INTERFACE ITF_BaseSaM

METHOD PUBLIC GetMode : E_BaseMachineMode
VAR_INPUT
END_VAR
END_METHOD

METHOD PUBLIC GetState : E_BaseMachineState
VAR_INPUT
END_VAR
END_METHOD

(*			
	EVERDE sp. z o.o.
	Rafał Osajda		25.10.2025		TC 4024.66
	Czy trwa zmianay trybu
*)
METHOD PUBLIC IsChangeModeBusy : BOOL
VAR_INPUT
END_VAR
END_METHOD

(*			
	EVERDE sp. z o.o.
	Rafał Osajda		25.10.2025		TC 4024.66
	Czy trwa zmiana stanu
*)
METHOD PUBLIC IsChangeStateBusy : BOOL
VAR_INPUT

END_VAR
END_METHOD

END_INTERFACE

(* stored: Version 1.1.0.1
   Itf ITF_BaseSaM: Id {e06ea4d8-10a4-07fe-0bda-c5cd43560d4e}
   Method GetMode: Id {17ad96f9-f8c6-06b4-06e2-cdfe42403acb}
   Method GetState: Id {d5368088-86fd-0411-1ca9-12bdae93bf00}
   Method IsChangeModeBusy: Id {0dd216ea-27b5-01b9-033f-72faa5a0d597}
   Method IsChangeStateBusy: Id {2bd79ff5-9782-015d-0a64-00caef1a80f6} *)
